FUNCTION_BLOCK ProductionServices (* Composite Function Block Type *)
  (* Standard: 61499-2 *)
  (* Version 0.0, 11/2/2020, prana, nxtControl GmbH, template *)
  PACKAGE Main;
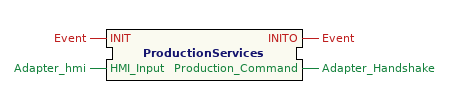
  EVENT_INPUT
    INIT; (* Initialization Request *)
  END_EVENT
  EVENT_OUTPUT
    INITO; (* Initialization Confirm *)
  END_EVENT
  SOCKETS
    HMI_Input : Adapter_hmi;
  END_SOCKETS
  PLUGS
    Production_Command : Adapter_Handshake;
  END_PLUGS
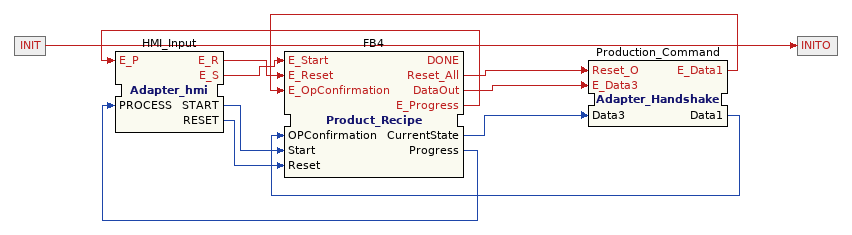
  FBS
    FB4 : Product_Recipe;
  END_FBS
  EVENT_CONNECTIONS
    INIT TO INITO;
    FB4.Reset_All TO Production_Command.Reset_O;
    FB4.DataOut TO Production_Command.E_Data3;
    Production_Command.E_Data1 TO FB4.E_OpConfirmation;
    HMI_Input.E_R TO FB4.E_Reset;
    FB4.E_Progress TO HMI_Input.E_P;
    HMI_Input.E_S TO FB4.E_Start;
  END_CONNECTIONS
  DATA_CONNECTIONS
    FB4.CurrentState TO Production_Command.Data3;
    Production_Command.Data1 TO FB4.OPConfirmation;
    FB4.Progress TO HMI_Input.PROCESS;
    HMI_Input.START TO FB4.Start;
    HMI_Input.RESET TO FB4.Reset;
  END_CONNECTIONS
END_FUNCTION_BLOCK
